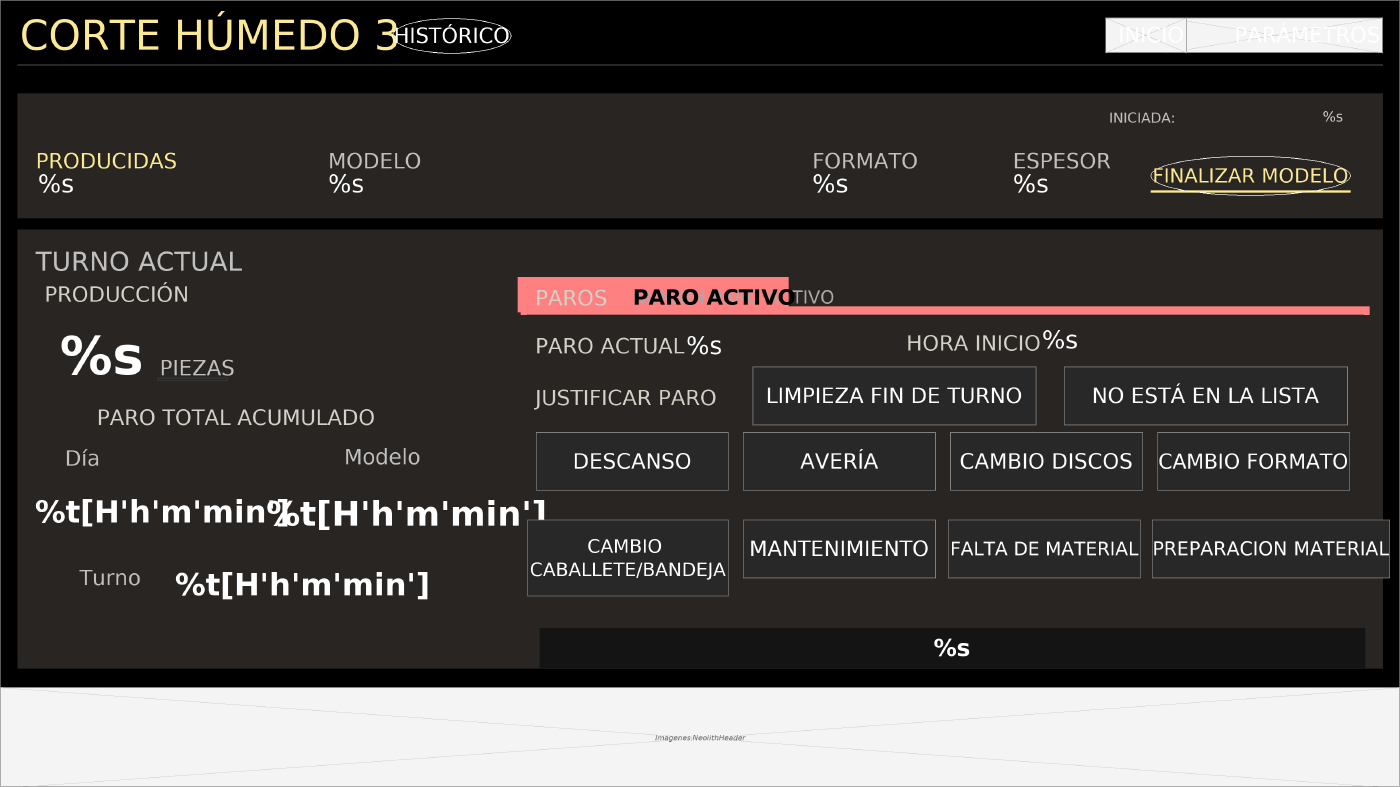
VISUALIZATION Home_CortH3  // 1920x1080
    Rectangle (24,315 1872x602)
    Rectangle (24,128 1872x171)
    Rectangle (24,88 1872x2)
    Label (24,16 514x64), "CORTE HÚMEDO 3"
    Rectangle (1426,451 183x30), "%s", text variable: FuncParoNodoLocalCorteH3.Funci_CortHum3.H_InParo_Ftc, invisible if: FuncParoNodoLocalCorteH3.Funci_CortHum3.M_SinParo_Ftc
    Rectangle (938,459 192x30), "%s", text variable: FuncParoNodoLocalCorteH3.Funci_CortHum3.Min_Parado_Ftc, invisible if: FuncParoNodoLocalCorteH3.Funci_CortHum3.M_SinParo_Ftc
    Rectangle (1573,147 272x27), "%s", text variable: FuncParoNodoLocalCorteH3.sFechaInicModeloTab
    Label (1518,147 99x30), "INICIADA:"
    Rectangle (740,862 1132x54), "%s", text variable: FuncParoNodoLocalCorteH3.Funci_CortHum3.S_Justi_Paro_Ftc, invisible if: FuncParoNodoLocalCorteH3.Funci_CortHum3.M_SinParo_Ftc, input disabled if: FuncParoNodoLocalCorteH3.FunGeneCortHum3.IndexJustificacionParo<>10
        OnMouseDown: write the text variable via Edit
    Image (1600,24 296x48), "PARÁMETROS"
        OnMouseClick: change screen: Ajustes_CorteH3
    Image (1516,24 111x48), "INICIO"
        OnMouseClick: change screen: Home_Sel_Maq
    Rectangle (447,232 671x40), "%s", text variable: FuncParoNodoLocalCorteH3.sModeloActualTabla, colour toggle: FuncParoNodoLocalCorteH3.Funci_CortHum3.Fotocelula
    Rectangle (1386,232 120x40), "%s", text variable: FuncParoNodoLocalCorteH3.FunGeneCortHum3.s_EspesorActualTabla
    Rectangle (1111,232 275x40), "%s", text variable: FuncParoNodoLocalCorteH3.FunGeneCortHum3.s_FormatoActualTabla
    Label (447,203 487x36), "MODELO"
    Label (1111,203 156x36), "FORMATO"
    Label (1386,203 156x36), "ESPESOR"
    Label (46,203 199x36), "PRODUCIDAS"
    Rectangle (49,232 248x40), "%s", text variable: FuncParoNodoLocalCorteH3.Funci_CortHum3.Cont_Piezas_Ftc
    Rectangle (1578,261 274x3)
    Ellipse (1578,214 274x54), "FINALIZAR MODELO"
        OnMouseClick: OpenDialog Dialog=V_Emerg_Fin_Prod_Ch3, OpenModal=True, OpenCentered=True
    Label (46,332 390x54), "TURNO ACTUAL"
    Label (58,386 199x36), "PRODUCCIÓN"
    Label (731,457 261x36), "PARO ACTUAL", invisible if: FuncParoNodoLocalCorteH3.Funci_CortHum3.M_SinParo_Ftc
    Label (1240,453 261x36), "HORA INICIO", invisible if: FuncParoNodoLocalCorteH3.Funci_CortHum3.M_SinParo_Ftc
    RoundedRectangle (735,593 264x80), "DESCANSO", invisible if: FuncParoNodoLocalCorteH3.Funci_CortHum3.M_SinParo_Ftc
        OnMouseClick: execute { FuncParoNodoLocalCorteH3.FunGeneCortHum3.IndexJustificacionParo:=1; FuncParoNodoLocalCorteH3.FunGeneCortHum3.ListadoJustificacionParo(); }
    RoundedRectangle (1019,593 264x80), "AVERÍA", invisible if: FuncParoNodoLocalCorteH3.Funci_CortHum3.M_SinParo_Ftc
        OnMouseClick: execute { FuncParoNodoLocalCorteH3.FunGeneCortHum3.IndexJustificacionParo:=2; FuncParoNodoLocalCorteH3.FunGeneCortHum3.ListadoJustificacionParo(); }
    RoundedRectangle (1303,593 264x80), "CAMBIO DISCOS", invisible if: FuncParoNodoLocalCorteH3.Funci_CortHum3.M_SinParo_Ftc
        OnMouseClick: execute { FuncParoNodoLocalCorteH3.FunGeneCortHum3.IndexJustificacionParo:=3; FuncParoNodoLocalCorteH3.FunGeneCortHum3.ListadoJustificacionParo(); }
    RoundedRectangle (1587,593 264x80), "CAMBIO FORMATO", invisible if: FuncParoNodoLocalCorteH3.Funci_CortHum3.M_SinParo_Ftc
        OnMouseClick: execute { FuncParoNodoLocalCorteH3.FunGeneCortHum3.IndexJustificacionParo:=4; FuncParoNodoLocalCorteH3.FunGeneCortHum3.ListadoJustificacionParo(); }
    Rectangle (79,444 183x88), "%s", text variable: FuncParoNodoLocalCorteH3.Funci_CortHum3.Cont_Piezas_Ftc
    Label (216,487 106x36), "PIEZAS"
    Rectangle (216,518 96x4), colour toggle: FuncParoNodoLocalCorteH3.Funci_CortHum3.Fotocelula
    Label (731,528 261x36), "JUSTIFICAR PARO", invisible if: FuncParoNodoLocalCorteH3.Funci_CortHum3.M_SinParo_Ftc
    Rectangle (714,424 1164x4), invisible if: FuncParoNodoLocalCorteH3.Funci_CortHum3.M_SinParo_Ftc
    Rectangle (710,380 371x48), invisible if: FuncParoNodoLocalCorteH3.Funci_CortHum3.M_SinParo_Ftc
    Label (731,391 199x36), "PAROS", invisible if: FuncParoNodoLocalCorteH3.Funci_CortHum3.M_SinParo_Ftc
    Label (865,393 326x30), "NINGÚN PARO ACTIVO", invisible if: FuncParoNodoLocalCorteH3.Funci_CortHum3.MParo_Ftc
    Label (865,393 235x30), "PARO ACTIVO", invisible if: FuncParoNodoLocalCorteH3.Funci_CortHum3.M_SinParo_Ftc
    Ellipse (538,25 163x48), "HISTÓRICO"
        OnMouseClick: change screen: HistTablaTablas_Ch2
    Label (130,555 367x36), "PARO TOTAL ACUMULADO"
    Rectangle (45,658 295x88), "%t[H'h'm'min']", text variable: FuncParoNodoLocalCorteH3.Funci_CortHum3.fbTiempParoAcumDiario.t_Acumulado
    Label (86,611 76x36), "Día"
    Image (-3,943 1927x139), image: Imagenes.NeolithHeader
    Rectangle (237,758 325x88), "%t[H'h'm'min']", text variable: FuncParoNodoLocalCorteH3.Funci_CortHum3.fbTiempParoAcumTurno.t_Acumulado
    Label (106,775 102x36), "Turno"
    Rectangle (362,661 388x88), "%t[H'h'm'min']", text variable: FuncParoNodoLocalCorteH3.Funci_CortHum3.fbTiempParoAcumModelo.t_Acumulado
    Label (469,609 118x36), "Modelo"
    RoundedRectangle (723,713 276x105), "CAMBIO CABALLETE/BANDEJA", invisible if: FuncParoNodoLocalCorteH3.Funci_CortHum3.M_SinParo_Ftc
        OnMouseClick: execute { FuncParoNodoLocalCorteH3.FunGeneCortHum3.IndexJustificacionParo:=5; FuncParoNodoLocalCorteH3.FunGeneCortHum3.ListadoJustificacionParo(); }
    RoundedRectangle (1019,713 264x80), "MANTENIMIENTO", invisible if: FuncParoNodoLocalCorteH3.Funci_CortHum3.M_SinParo_Ftc
        OnMouseClick: execute { FuncParoNodoLocalCorteH3.FunGeneCortHum3.IndexJustificacionParo:=6; FuncParoNodoLocalCorteH3.FunGeneCortHum3.ListadoJustificacionParo(); }
    RoundedRectangle (1300,713 264x80), "FALTA DE MATERIAL", invisible if: FuncParoNodoLocalCorteH3.Funci_CortHum3.M_SinParo_Ftc
        OnMouseClick: execute { FuncParoNodoLocalCorteH3.FunGeneCortHum3.IndexJustificacionParo:=7; FuncParoNodoLocalCorteH3.FunGeneCortHum3.ListadoJustificacionParo(); }
    RoundedRectangle (1580,713 326x80), "PREPARACION MATERIAL", invisible if: FuncParoNodoLocalCorteH3.Funci_CortHum3.M_SinParo_Ftc
        OnMouseClick: execute { FuncParoNodoLocalCorteH3.FunGeneCortHum3.IndexJustificacionParo:=8; FuncParoNodoLocalCorteH3.FunGeneCortHum3.ListadoJustificacionParo(); }
    RoundedRectangle (1032,503 389x80), "LIMPIEZA FIN DE TURNO", invisible if: FuncParoNodoLocalCorteH3.Funci_CortHum3.M_SinParo_Ftc
        OnMouseClick: execute { FuncParoNodoLocalCorteH3.FunGeneCortHum3.IndexJustificacionParo:=9; FuncParoNodoLocalCorteH3.FunGeneCortHum3.ListadoJustificacionParo(); }
    RoundedRectangle (1459,503 389x80), "NO ESTÁ EN LA LISTA", invisible if: FuncParoNodoLocalCorteH3.Funci_CortHum3.M_SinParo_Ftc
        OnMouseClick: execute { FuncParoNodoLocalCorteH3.FunGeneCortHum3.IndexJustificacionParo:=10; FuncParoNodoLocalCorteH3.FunGeneCortHum3.ListadoJustificacionParo(); }
END_VISUALIZATION

(* stored: Version 1.1.0.1, ProductVersion 3.1.4024.12
   Visu Home_CortH3: Id {9e281147-de25-4bb2-8a2f-652225f7024c} *)
